TYPE ST_HeatingNetworkHighTemperatureControl :
STRUCT
	fFeedTemperature : REAL;
	fTargetTemperature : REAL;
	bAlgorithmPermission : BOOL;
	bSetStatusOn_CHP1 : BOOL;
	bSetStatusOn_CHP2 : BOOL;
	bSetStatusOn_CondensingBoiler : BOOL;
	bSetStatusOn_StaticHeating : BOOL;
	bSetStatusOn_VSIStorage : BOOL;
	bLoading_VSISystem : BOOL;
END_STRUCT
END_TYPE

(* stored: Version 1.1.0.1, ProductVersion 3.1.4024.10
   DUT ST_HeatingNetworkHighTemperatureControl: Id {62265abc-da42-46bc-b58c-32abc31e7390} *)
